Staubli VAL3: stop.pgx

program stop()
begin
  logMsg("ros2_server::stop : quitting application")
  // Stop motion
  stopMove()
  resetMotion()
  // Clear socket buffers
  clearBuffer(siSocketControl)
end
